TYPE TYP_VALVE_53_HW :
STRUCT
	In : TYP_VALVE_53_HW_IN;
	Out : TYP_VALVE_53_HW_OUT;
END_STRUCT
END_TYPE

(* stored: Version 1.1.0.1, ProductVersion 3.1.4024.12
   DUT TYP_VALVE_53_HW: Id {25582c25-1c57-4bc9-a0f7-1b61f0b5ceeb} *)
